Staubli VAL3: removePart.pgx

public program removePart(num x_nConvNum (dimensions=1))
begin
  // This program deletes the first object in the queue. The part will
  //  not be deleted until all command tracking movements associated
  //  to this part have been executed by the robot arm.
  //
  // Input Param
  //  x_nConvNum : Conveyor number
  //
  // Output param
  //  none       :
  //
  //----------------------------------------------------------------
  //
  if cfg:bLog
    logMsg("MOT(removePart)>>Request to remove part from queue of conveyor "+toString("",x_nConvNum))
  endIf
  switch x_nConvNum
    case 0
      call cnv0:removePart()
    break
    case 1
      call cnv1:removePart()
    break
  endSwitch
end
